(* PLC project Sin nombre, Desconocido Sin nombre 1 *)
(* stored: creationDateTime 2020-09-23T19:30:14, modificationDateTime 2025-06-17T16:05:16 *)

PROGRAM program0
  VAR
    FC_CERRADA : BOOL;
    FC_BYPASS : BOOL;
    FC_ABIERTA : BOOL;
    Apertura : BOOL;
    Pausa : BOOL;
    Cierre : BOOL;
    Q_BOMBA : BOOL;
    Q_VALV_CIERRE : BOOL;
    PASO_1 : BOOL;
    PASO_2 : BOOL;
    PASO_3 : BOOL;
    PASO_4 : BOOL;
    PASO_5 : BOOL;
    PASO_6 : BOOL;
    Temp_Apertura : TON;
    Temp_Bloqueo : TON;
    Temp_Rearranque : TON;
  END_VAR
  VAR  (* added by the conversion: wires and edge detectors of the diagram *)
    R_TRIG1 : R_TRIG;
  END_VAR

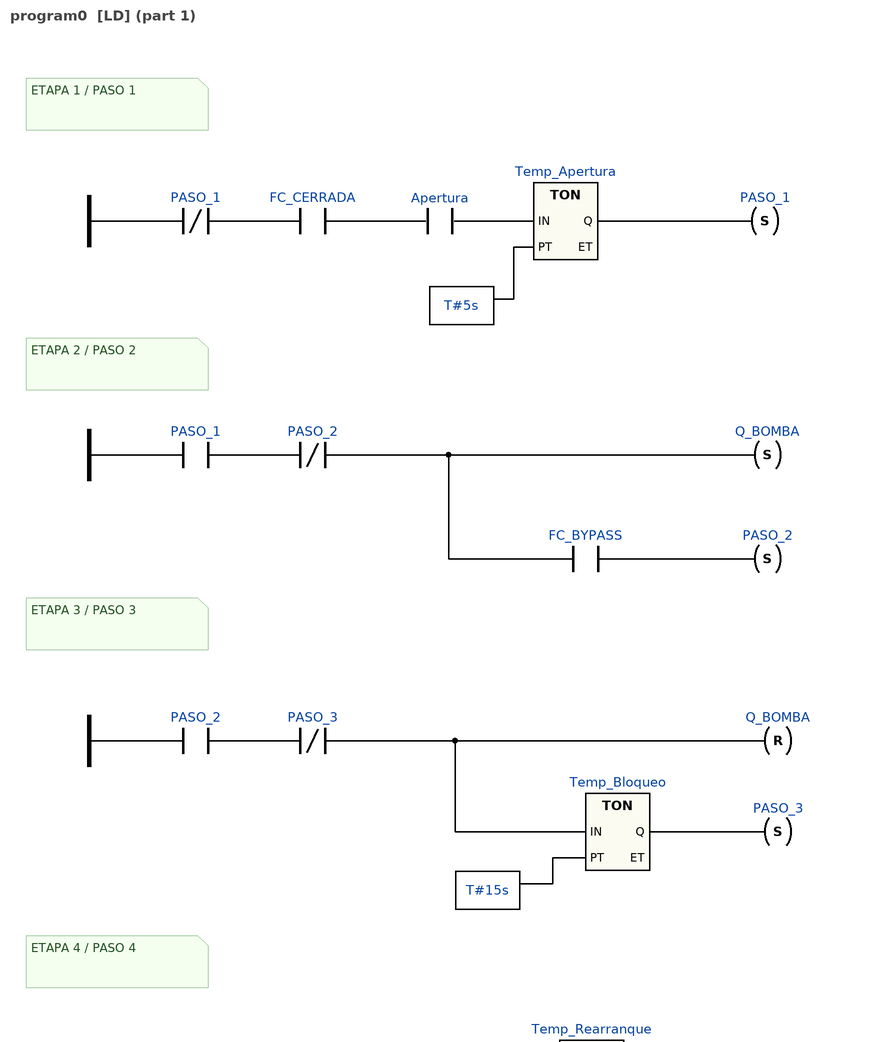
(* LD diagram, written out as Structured Text *)
(* ETAPA 1 / PASO 1 *)
Temp_Apertura(IN := NOT PASO_1 AND FC_CERRADA AND Apertura, PT := T#5s);
IF Temp_Apertura.Q THEN PASO_1 := TRUE; END_IF;
(* ETAPA 2 / PASO 2 *)
IF PASO_1 AND NOT PASO_2 THEN Q_BOMBA := TRUE; END_IF;
IF PASO_1 AND NOT PASO_2 AND FC_BYPASS THEN PASO_2 := TRUE; END_IF;
(* ETAPA 3 / PASO 3 *)
IF PASO_2 AND NOT PASO_3 THEN Q_BOMBA := FALSE; END_IF;
Temp_Bloqueo(IN := PASO_2 AND NOT PASO_3, PT := T#15s);
IF Temp_Bloqueo.Q THEN PASO_3 := TRUE; END_IF;
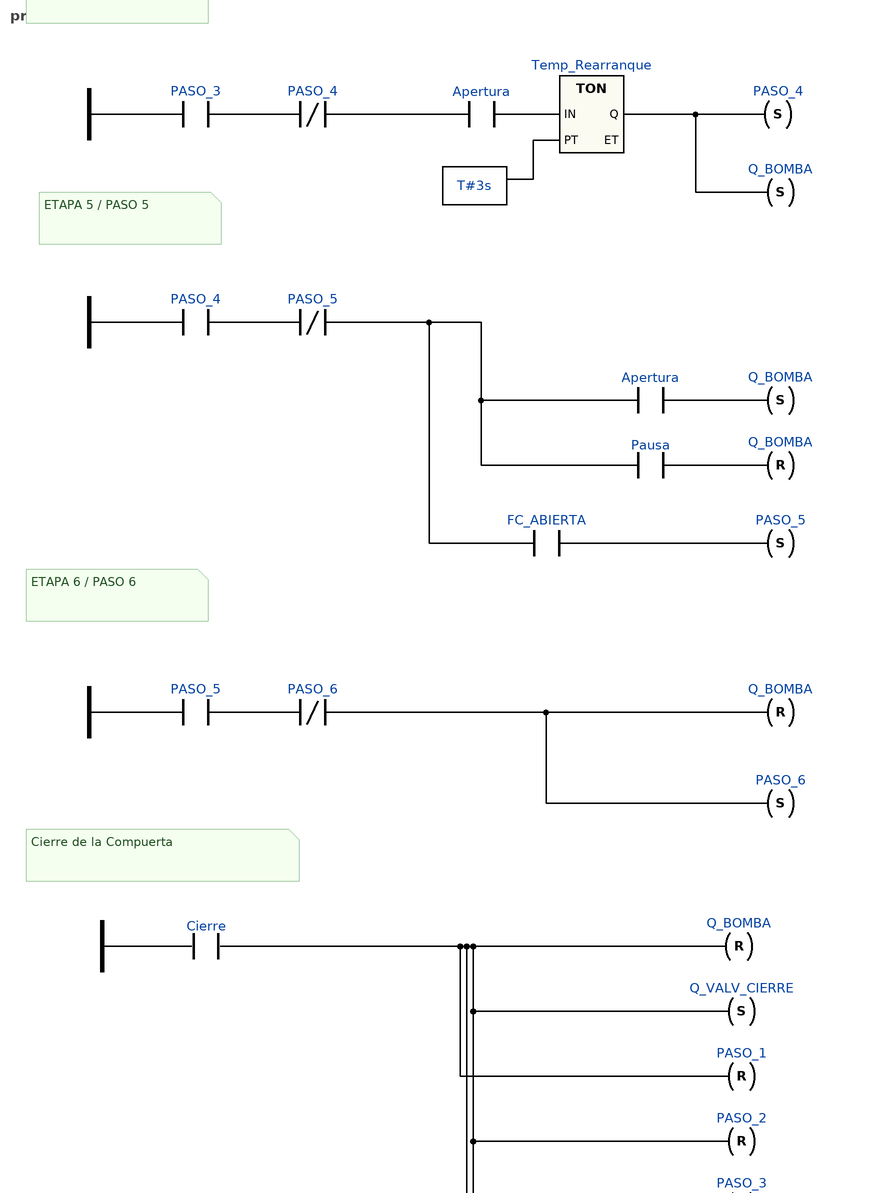
(* ETAPA 4 / PASO 4 *)
Temp_Rearranque(IN := PASO_3 AND NOT PASO_4 AND Apertura, PT := T#3s);
IF Temp_Rearranque.Q THEN PASO_4 := TRUE; END_IF;
(* ETAPA 5 / PASO 5 *)
IF PASO_4 AND NOT PASO_5 AND Apertura THEN Q_BOMBA := TRUE; END_IF;
IF PASO_4 AND NOT PASO_5 AND Pausa THEN Q_BOMBA := FALSE; END_IF;
IF PASO_4 AND NOT PASO_5 AND FC_ABIERTA THEN PASO_5 := TRUE; END_IF;
(* ETAPA 6 / PASO 6 *)
IF PASO_5 AND NOT PASO_6 THEN Q_BOMBA := FALSE; END_IF;
IF PASO_5 AND NOT PASO_6 THEN PASO_6 := TRUE; END_IF;
(* Cierre de la Compuerta *)
IF Cierre THEN Q_BOMBA := FALSE; END_IF;
IF Cierre THEN Q_VALV_CIERRE := TRUE; END_IF;
IF Cierre THEN PASO_1 := FALSE; END_IF;
IF Cierre THEN PASO_2 := FALSE; END_IF;
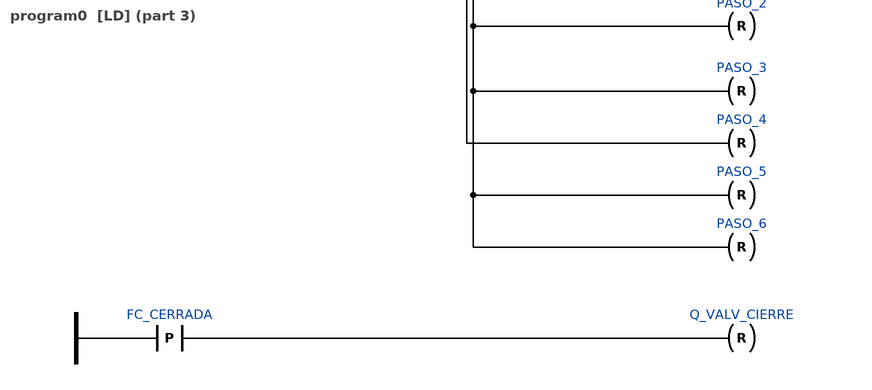
IF Cierre THEN PASO_3 := FALSE; END_IF;
IF Cierre THEN PASO_4 := FALSE; END_IF;
IF Cierre THEN PASO_5 := FALSE; END_IF;
IF Cierre THEN PASO_6 := FALSE; END_IF;
R_TRIG1(CLK := FC_CERRADA);
IF R_TRIG1.Q THEN Q_VALV_CIERRE := FALSE; END_IF;
IF Temp_Rearranque.Q THEN Q_BOMBA := TRUE; END_IF;
END_PROGRAM

CONFIGURATION Config0
  RESOURCE Res0 ON PLC
    TASK task0(INTERVAL := T#20ms, PRIORITY := 0);
    PROGRAM instance0 WITH task0 : program0;
  END_RESOURCE
END_CONFIGURATION
